(* PLC project  *)

PROGRAM P
  VAR  (* added by the conversion: wires and edge detectors of the diagram *)
    _ADD3_ENO : BOOL;
    _ADD3_OUT : ANY;
    _ADD13_ENO : BOOL;
    _ADD13_OUT : ANY;
  END_VAR

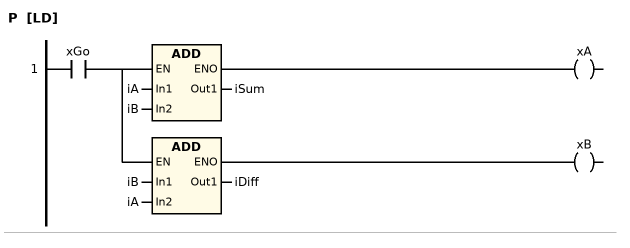
(* LD diagram, written out as Structured Text *)
_ADD3_OUT := ADD(EN := xGo, IN1 := iA, IN2 := iB, ENO => _ADD3_ENO);
xA := _ADD3_ENO;
IF _ADD3_ENO THEN iSum := _ADD3_OUT; END_IF;
_ADD13_OUT := ADD(EN := xGo, IN1 := iB, IN2 := iA, ENO => _ADD13_ENO);
xB := _ADD13_ENO;
IF _ADD13_ENO THEN iDiff := _ADD13_OUT; END_IF;
END_PROGRAM
